(* IEC 61131-3 sources: 2026_Projet_YGO_ExcavatriceDragage/CODE/CONTROL, 3 files *)

(* ---- PRG_6_WinchControl.st ---- *)
(* ═══════════════════════════════════════════════════════════════
   🪝 PRG_6_WinchControl — Commande des Treuils M1/M2, Synchro et Grappin
   ───────────────────────────────────────────────────────────────
   ⚙️ Exécuté par la tâche PLC en position 6.
   ✅ Arbitre entre les commandes Manuelles (Joystick) et Automatiques (PRG_5_Cycle).
   ═══════════════════════════════════════════════════════════════ *)

PROGRAM PRG_6_WinchControl
VAR
    // Stubs
    StubMachineEnableN1 : BOOL := TRUE;

    // Instances
    instWinchSync : FB_WinchSync;
    instGrappin   : FB_Grappin;
    instWinchM1   : FB_Winch;
    instWinchM2   : FB_Winch;

    // Variables de commande M1 après arbitrage Manuel/Auto
    M1_StartStop_Active     : BOOL;
    M1_Direction_Active     : INT;
    M1_SpeedRef_Active      : REAL;

    // Variables de commande M2 après arbitrage Grappin/Manuel/Auto
    M2_StartStop_Active     : BOOL;
    M2_Direction_Active     : INT;
    M2_SpeedRef_Active      : REAL;
    M2_SpeedStepTableActive : ST_SpeedStepTable;

    // Bornage et limites
    BottomLimitM1_Active    : REAL;
    BottomLimitM2_Active    : REAL;
    ForbidDescentM1_Active  : BOOL;
    ForbidDescentM2_Active  : BOOL;
END_VAR

// === IMPLEMENTATION (corps du PROGRAM PRG_6_WinchControl) ===

// ── 1. ARBITRAGE DES CONSIGNES M1 (Joystick vs Cycle Automatique) ────────
IF PRG_4_Modes.instModes.Mode = E_Mode.SEMI_AUTO THEN
    M1_StartStop_Active := PRG_5_Cycle.instCycle.CmdWinchM1_StartStop;
    M1_Direction_Active := PRG_5_Cycle.instCycle.CmdWinchM1_Direction;
    M1_SpeedRef_Active  := PRG_5_Cycle.instCycle.CmdWinchM1_SpeedPct;
ELSE
    M1_StartStop_Active := PRG_1_Diagnostics.FB_Joystick_0.AxisCmdY.StartStop AND NOT instGrappin.Busy;
    M1_Direction_Active := PRG_1_Diagnostics.FB_Joystick_0.AxisCmdY.Direction;
    M1_SpeedRef_Active  := PRG_1_Diagnostics.FB_Joystick_0.AxisCmdY.SpeedRef;
END_IF;

// ── 2. ARBITRAGE DES CONSIGNES M2 (Grappin vs Cycle Automatique vs Joystick) ──
IF instGrappin.Busy THEN
    M2_StartStop_Active := instGrappin.M2_StartStop;
    M2_Direction_Active := instGrappin.M2_Direction;
    M2_SpeedRef_Active  := 15.0; // Vitesse lente forcée pour fermeture grappin
ELSE
    IF PRG_4_Modes.instModes.Mode = E_Mode.SEMI_AUTO THEN
        M2_StartStop_Active := PRG_5_Cycle.instCycle.CmdWinchM2_StartStop;
        M2_Direction_Active := PRG_5_Cycle.instCycle.CmdWinchM2_Direction;
        M2_SpeedRef_Active  := PRG_5_Cycle.instCycle.CmdWinchM2_SpeedPct;
    ELSE
        M2_StartStop_Active := PRG_1_Diagnostics.FB_Joystick_0.AxisCmdY.StartStop;
        M2_Direction_Active := PRG_1_Diagnostics.FB_Joystick_0.AxisCmdY.Direction;
        M2_SpeedRef_Active  := PRG_1_Diagnostics.FB_Joystick_0.AxisCmdY.SpeedRef;
    END_IF;
END_IF;

// ── 3. SURVEILLANCE ÉCART DE SYNCHRONISATION ────────────────────────────
instWinchSync(
    Enable          := NOT PRG_4_Modes.instModes.OverrideSync AND NOT instGrappin.Busy,
    Reset           := PRG_9_Supervision.MachineReset_IHM,
    EmergencyStopOk := PRG_0_Inputs.EmergencyStopOk,
    Mode            := PRG_4_Modes.instModes.Mode,
    CablePosM1      := PRG_2_Encoders.instEncoderScaleM1.CablePosM,
    CablePosM2      := PRG_2_Encoders.instEncoderScaleM2.CablePosM,
    HomedM1         := PRG_2_Encoders.instHomingM1.Homed,
    HomedM2         := PRG_2_Encoders.instHomingM2.Homed,
    OverrideSync    := PRG_4_Modes.instModes.OverrideSync,
    SyncToleranceM  := GVL_PERSISTENT.WinchSyncTolerance_M,
    ActiveOffsetM   := instGrappin.ActiveOffsetM,

    RelayFwdM1      := instWinchM1.RelayFwd,
    RelayFwdM2      := instWinchM2.RelayFwd,
    RelayRevM1      := instWinchM1.RelayRev,
    RelayRevM2      := instWinchM2.RelayRev,
    Contactor1_M1   := instWinchM1.Contactor1,
    Contactor1_M2   := instWinchM2.Contactor1,
    Contactor2_M1   := instWinchM1.Contactor2,
    Contactor2_M2   := instWinchM2.Contactor2,
    Contactor3_M1   := instWinchM1.Contactor3,
    Contactor3_M2   := instWinchM2.Contactor3,
    Contactor4_M1   := instWinchM1.Contactor4,
    Contactor4_M2   := instWinchM2.Contactor4
);

// ── 4. COMMANDE DU GRAPPIN (Séquence lente) ─────────────────────────────
instGrappin(
    Enable              := TRUE,
    Reset               := PRG_9_Supervision.MachineReset_IHM,
    EmergencyStopOk     := PRG_0_Inputs.EmergencyStopOk,
    Mode                := PRG_4_Modes.instModes.Mode,
    CmdOpen_IHM         := GVL_IHM.Grappin.CmdOpen OR PRG_5_Cycle.instCycle.CmdGrappin_Open,
    CmdClose_IHM        := GVL_IHM.Grappin.CmdClose OR PRG_5_Cycle.instCycle.CmdGrappin_Close,
    JoystickY_StartStop := PRG_1_Diagnostics.FB_Joystick_0.AxisCmdY.StartStop,
    JoystickY_Direction := PRG_1_Diagnostics.FB_Joystick_0.AxisCmdY.Direction,
    CablePosM1          := PRG_2_Encoders.instEncoderScaleM1.CablePosM,
    CablePosM2          := PRG_2_Encoders.instEncoderScaleM2.CablePosM,
    Config              := GVL_PERSISTENT.GrappinConfig,
    TimeoutDuration     := GVL_IHM.Grappin.TimeoutDuration,
    GrappinState        := GVL_PERSISTENT.GrappinState
);

// Table active M2 (court-circuite les contacteurs si vitesse lente requise pour le grappin)
IF instGrappin.M2_ForceSlowSpeed THEN
    M2_SpeedStepTableActive.P1R1 := FALSE; M2_SpeedStepTableActive.P1R2 := FALSE; M2_SpeedStepTableActive.P1R3 := FALSE; M2_SpeedStepTableActive.P1R4 := FALSE;
    M2_SpeedStepTableActive.P2R1 := FALSE; M2_SpeedStepTableActive.P2R2 := FALSE; M2_SpeedStepTableActive.P2R3 := FALSE; M2_SpeedStepTableActive.P2R4 := FALSE;
    M2_SpeedStepTableActive.P3R1 := FALSE; M2_SpeedStepTableActive.P3R2 := FALSE; M2_SpeedStepTableActive.P3R3 := FALSE; M2_SpeedStepTableActive.P3R4 := FALSE;
    M2_SpeedStepTableActive.P4R1 := FALSE; M2_SpeedStepTableActive.P4R2 := FALSE; M2_SpeedStepTableActive.P4R3 := FALSE; M2_SpeedStepTableActive.P4R4 := FALSE;
    M2_SpeedStepTableActive.P5R1 := FALSE; M2_SpeedStepTableActive.P5R2 := FALSE; M2_SpeedStepTableActive.P5R3 := FALSE; M2_SpeedStepTableActive.P5R4 := FALSE;
    M2_SpeedStepTableActive.StepThreshold_Pct := GVL_PERSISTENT.WinchM2SpeedStepTable.StepThreshold_Pct;
ELSE
    M2_SpeedStepTableActive := GVL_PERSISTENT.WinchM2SpeedStepTable;
END_IF;

// ── 5. CALCUL DES LIMITES BASSES ACTIVES ET DU BLOCAGE DE DESCENTE ──────
BottomLimitM1_Active := GVL_PERSISTENT.CableLimitDescent_M;
IF (PRG_4_Modes.instModes.Mode = E_Mode.SEMI_AUTO) AND GVL_PERSISTENT.LimitLegalEnabled THEN
    BottomLimitM1_Active := MAX(BottomLimitM1_Active, GVL_PERSISTENT.LimitLegalDepthMinAllowed);
END_IF;

BottomLimitM2_Active := GVL_PERSISTENT.CableLimitDescent_M;
IF (PRG_4_Modes.instModes.Mode = E_Mode.SEMI_AUTO) AND GVL_PERSISTENT.LimitLegalEnabled THEN
    BottomLimitM2_Active := MAX(BottomLimitM2_Active, GVL_PERSISTENT.LimitLegalDepthMinAllowed);
END_IF;

ForbidDescentM1_Active := PRG_3_Safety.instSafetyWinchM1.ForbidDescent
                          OR ((PRG_4_Modes.instModes.Mode = E_Mode.SEMI_AUTO)
                              AND GVL_PERSISTENT.LimitLegalEnabled
                              AND (PRG_2_Encoders.instEncoderScaleM1.CablePosM <= GVL_PERSISTENT.LimitLegalDepthMinAllowed));

ForbidDescentM2_Active := PRG_3_Safety.instSafetyWinchM2.ForbidDescent
                          OR ((PRG_4_Modes.instModes.Mode = E_Mode.SEMI_AUTO)
                              AND GVL_PERSISTENT.LimitLegalEnabled
                              AND (PRG_2_Encoders.instEncoderScaleM2.CablePosM <= GVL_PERSISTENT.LimitLegalDepthMinAllowed));

// ── 6. EXÉCUTION DU PILOTAGE DU TREUIL M1 ───────────────────────────────
instWinchM1(
    Enable                  := StubMachineEnableN1,
    Reset                   := PRG_9_Supervision.MachineReset_IHM,
    EmergencyStopOk         := PRG_0_Inputs.EmergencyStopOk,
    Mode                    := PRG_4_Modes.instModes.Mode,
    StartStop               := M1_StartStop_Active,
    SafeStop                := PRG_3_Safety.instSafetyWinchM1.SafeStop OR ((instWinchSync.ErrorId AND 16#0002) <> 16#0000),
    ForbidDescent           := ForbidDescentM1_Active,
    ForbidAscent            := PRG_3_Safety.instSafetyWinchM1.ForbidAscent,
    Direction               := M1_Direction_Active,
    SpeedRefPct             := M1_SpeedRef_Active,
    SpeedStepTable          := GVL_PERSISTENT.WinchM1SpeedStepTable,
    MaxStepDescente         := GVL_PERSISTENT.WinchM1MaxStepDescente,
    ContactorFeedbackFwd    := PRG_0_Inputs.M1ContactorFeedbackFwd,
    ContactorFeedbackRev    := PRG_0_Inputs.M1ContactorFeedbackRev,
    BrakeFeedback           := PRG_0_Inputs.M1BrakeFeedback,
    RampAccelRate           := GVL_PERSISTENT.WinchM1RampAccelRate_Pct,
    RampDecelNormalRate     := GVL_PERSISTENT.WinchM1RampDecelNormal_Pct,
    RampDecelFastRate       := GVL_PERSISTENT.WinchM1RampDecelFast_Pct,
    Homed                   := PRG_2_Encoders.instHomingM1.Homed,
    CablePosM               := PRG_2_Encoders.instEncoderScaleM1.CablePosM,
    TopLimitM               := GVL_PERSISTENT.HomingTargetM1_M,
    BottomLimitM            := BottomLimitM1_Active,
    SlowdownDistanceM       := GVL_PERSISTENT.WinchSlowdownDistance_M,
    SlowSpeedPct            := GVL_PERSISTENT.WinchSlowSpeedPct
);

// ── 7. EXÉCUTION DU PILOTAGE DU TREUIL M2 ───────────────────────────────
instWinchM2(
    Enable                  := StubMachineEnableN1,
    Reset                   := PRG_9_Supervision.MachineReset_IHM,
    EmergencyStopOk         := PRG_0_Inputs.EmergencyStopOk,
    Mode                    := PRG_4_Modes.instModes.Mode,
    StartStop               := M2_StartStop_Active,
    SafeStop                := PRG_3_Safety.instSafetyWinchM2.SafeStop OR ((instWinchSync.ErrorId AND 16#0002) <> 16#0000),
    ForbidDescent           := ForbidDescentM2_Active,
    ForbidAscent            := PRG_3_Safety.instSafetyWinchM2.ForbidAscent,
    Direction               := M2_Direction_Active,
    SpeedRefPct             := M2_SpeedRef_Active,
    SpeedStepTable          := M2_SpeedStepTableActive,
    MaxStepDescente         := GVL_PERSISTENT.WinchM2MaxStepDescente,
    ContactorFeedbackFwd    := PRG_0_Inputs.M2ContactorFeedbackFwd,
    ContactorFeedbackRev    := PRG_0_Inputs.M2ContactorFeedbackRev,
    BrakeFeedback           := PRG_0_Inputs.M2BrakeFeedback,
    RampAccelRate           := GVL_PERSISTENT.WinchM2RampAccelRate_Pct,
    RampDecelNormalRate     := GVL_PERSISTENT.WinchM2RampDecelNormal_Pct,
    RampDecelFastRate       := GVL_PERSISTENT.WinchM2RampDecelFast_Pct,
    Homed                   := PRG_2_Encoders.instHomingM2.Homed,
    CablePosM               := PRG_2_Encoders.instEncoderScaleM2.CablePosM,
    TopLimitM               := GVL_PERSISTENT.HomingTargetM2_M,
    BottomLimitM            := BottomLimitM2_Active,
    SlowdownDistanceM       := GVL_PERSISTENT.WinchSlowdownDistance_M,
    SlowSpeedPct            := GVL_PERSISTENT.WinchSlowSpeedPct
);

(* ---- PRG_7_ChariotControl.st ---- *)
(* ═══════════════════════════════════════════════════════════════
   ↔️ PRG_7_ChariotControl — Pilotage de la Translation Chariot M3
   ───────────────────────────────────────────────────────────────
   ⚙️ Exécuté par la tâche PLC en position 7.
   ✅ Arbitre entre les commandes Manuelles (Joystick) et Automatiques (PRG_5_Cycle).
   ═══════════════════════════════════════════════════════════════ *)

PROGRAM PRG_7_ChariotControl
VAR
    instChariotM3           : FB_Chariot;

    // Commandes arbitrées après sélection Manuel/Auto
    M3_StartStop_Active     : BOOL;
    M3_Direction_Active     : INT;
    M3_SpeedRef_Active      : REAL;
    M3_PositionSensorTarget : BOOL;

    // Target active (HMI en manuel, instCycle en auto)
    SelectedTargetNum       : INT;
END_VAR

// === IMPLEMENTATION (corps du PROGRAM PRG_7_ChariotControl) ===

// ── 1. ARBITRAGE DU SÉLECTEUR DE CIBLE ET DE LA DIRECTION ──────────────────
IF PRG_4_Modes.instModes.Mode = E_Mode.SEMI_AUTO OR PRG_4_Modes.instModes.Mode = E_Mode.AUTO THEN
    // Mode Auto/Semi-Auto : Consigne issue du séquenceur de cycle
    SelectedTargetNum    := PRG_5_Cycle.instCycle.CmdChariotM3_Target;
    M3_StartStop_Active  := PRG_5_Cycle.instCycle.CmdChariotM3_Start;
    M3_SpeedRef_Active   := 40.0; // Vitesse de translation automatique nominale (40%)

    // Détermination automatique du sens de marche selon la cible :
    // - Trémie (cible 4) = Marche Avant (Direction := 1)
    // - Fosses (cible 1 et 2) = Marche Arrière (Direction := -1)
    IF SelectedTargetNum = 4 THEN
        M3_Direction_Active := 1;
    ELSE
        M3_Direction_Active := -1;
    END_IF;
ELSE
    // Mode Manuel/Maintenance : Consignes issues du Joystick et sélecteur HMI
    SelectedTargetNum    := StubChariotPositionSelect_IHM;
    M3_StartStop_Active  := PRG_1_Diagnostics.FB_Joystick_0.AxisCmdX.StartStop;
    M3_Direction_Active  := PRG_1_Diagnostics.FB_Joystick_0.AxisCmdX.Direction;
    M3_SpeedRef_Active   := PRG_1_Diagnostics.FB_Joystick_0.AxisCmdX.SpeedRef;
END_IF;

// Câblage du capteur de butée de la cible sélectionnée
CASE SelectedTargetNum OF
    1: M3_PositionSensorTarget := PRG_0_Inputs.ChariotPosFosse1;
    2: M3_PositionSensorTarget := PRG_0_Inputs.ChariotPosFosse2;
    3: M3_PositionSensorTarget := PRG_0_Inputs.ChariotPosMaintenance;
    4: M3_PositionSensorTarget := PRG_0_Inputs.ChariotPosTremie;
ELSE
    M3_PositionSensorTarget := FALSE;   // Aucun capteur visé
END_CASE;

// ── 2. EXÉCUTION DU PILOTAGE DU CHARIOT M3 ──────────────────────────────
instChariotM3(
    Enable                  := PRG_6_WinchControl.StubMachineEnableN1,
    Reset                   := PRG_9_Supervision.MachineReset_IHM,
    EmergencyStopOk         := PRG_0_Inputs.EmergencyStopOk,
    Mode                    := PRG_4_Modes.instModes.Mode,
    StartStop               := M3_StartStop_Active,
    SafeStop                := PRG_3_Safety.instSafetyChariotM3.SafeStop,
    CommMode                := E_ChariotCommMode.DEGRADED_IO,
    Direction               := M3_Direction_Active,
    SpeedRefPct             := M3_SpeedRef_Active,
    PositionSensorTarget    := M3_PositionSensorTarget,
    DriveStatusWord         := 0,
    DriveActualFreqHz       := 0.0,
    ContactorFeedbackFwd    := M3_ContactorFeedbackFwd,
    ContactorFeedbackRev    := M3_ContactorFeedbackRev,
    DriveFaultFeedback      := M3_DriveFaultFeedback,
    BrakeFeedback           := SEL(GVL_IHM.Chariot.BypassBrakeFeedback, PRG_0_Inputs.M3BrakeFeedback, instChariotM3.BrakeCmd)
);

// ── 3. RECOPIE VERS LES VARIABLES GLOBALES DE SIMULATION / STUBS ─────────
M3_RelayFwd     := instChariotM3.RelayFwd;
M3_RelayRev     := instChariotM3.RelayRev;
M3_RelaySpeedGv := instChariotM3.RelaySpeedGv;

M3_ContactorFeedbackFwd := M3_RelayFwd;
M3_ContactorFeedbackRev := M3_RelayRev;

(* ---- PRG_8_AuxiliaryControl.st ---- *)
(* ═══════════════════════════════════════════════════════════════
   ⚡ PRG_8_AuxiliaryControl — Gestion des Auxiliaires (Hydraulique, Crible...)
   ───────────────────────────────────────────────────────────────
   ⚙️ Exécuté par la tâche PLC en position 8.
   ✅ Regroupe toutes les commandes et logiques hors-axes.
   ═══════════════════════════════════════════════════════════════ *)

PROGRAM PRG_8_AuxiliaryControl
VAR
    // 🌡️ Groupe Hydraulique
    HydraulicPumpRunCmd   : BOOL;   // Commande démarrage centrale hydraulique
    HydraulicFaultOk      : BOOL;   // Retour défaut groupe hydraulique (NC)

    // 🌾 Crible (Sifter / Sieve)
    SifterRunCmd          : BOOL;   // Commande marche crible
    SifterFaultOk         : BOOL;   // Retour défaut électrique crible (NC)

    // 🔗 Divers
    GridOpenCmd           : BOOL;   // Commande ouverture grille
    HelmetCloseCmd        : BOOL;   // Commande fermeture casque
END_VAR

// === IMPLEMENTATION (corps du PROGRAM PRG_8_AuxiliaryControl) ===

// --- STUBS LOGIQUES TEMPORAIRES (comportement passif / neutre) ---
HydraulicPumpRunCmd := FALSE;
SifterRunCmd        := FALSE;
GridOpenCmd         := FALSE;
HelmetCloseCmd      := FALSE;

HydraulicFaultOk    := TRUE; // Par défaut sain (NC)
SifterFaultOk       := TRUE; // Par défaut sain (NC)
